(* CODESYS project Лабораторная работа №1.project

Project tree, tasks and I/O mapping:
  Device : CODESYS Control Win V3, 3S - Smart Software Solutions GmbH, order no. 305021, version 3.5.5.50
    application Application
      libraries: Standard, * (System)
      task MainTask (cyclic, interval t#20ms, priority 1) calls PLC_PRG
      task VISU_TASK (cyclic, interval 100 ms, priority 31) calls VisuElems.Visu_Prg
      program PLC_PRG [ST]
      global variables GVL
      visualisation Visualization
  text list GlobalTextList
*)

// Device/Application/GVL
VAR_GLOBAL
	upper_level_sensor: BOOL := FALSE;
	lower_level_sensor: BOOL := FALSE;
	
	pump_relay: BOOL := FALSE;
	yellow_lamp: BOOL := FALSE;
	green_lamp: BOOL := TRUE;
END_VAR

// Device/Application/PLC_PRG
PROGRAM PLC_PRG
VAR
	is_pumping: BOOL := FALSE;
END_VAR

// запускать/останавливать откачку 
// только при срабатывании сенсора
IF upper_level_sensor THEN
	is_pumping := TRUE;
ELSIF lower_level_sensor THEN
	is_pumping := FALSE;
END_IF

// если откачка запущена/остановлена,
// но реле ещё не сработало/отключено,
// то включить/отключить реле и нужную лампочку
IF is_pumping AND NOT pump_relay THEN
	pump_relay := TRUE;
	yellow_lamp := TRUE;
	green_lamp := FALSE;
ELSIF NOT is_pumping AND pump_relay THEN
	pump_relay := FALSE;
	yellow_lamp := FALSE;
	green_lamp := TRUE;
END_IF

END_PROGRAM

// Device/Application/Visualization
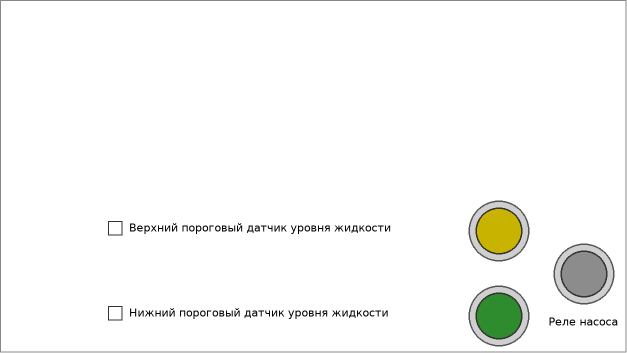
VISUALIZATION Visualization  // 627x353
    Checkbox (106,216 294x24), "Верхний пороговый датчик уровня жидкости", variable: upper_level_sensor
    Checkbox (106,301 294x24), "Нижний пороговый датчик уровня жидкости", variable: lower_level_sensor
    Group (464,196 70x155)
        Lamp1 (0,0 70x70), variable: yellow_lamp, style: Lamp-Lamp1-Yellow
        Lamp1 (0,85 70x70), variable: green_lamp, style: Lamp-Lamp1-Green
    Lamp1 (549,239 70x70), variable: pump_relay, style: Lamp-Lamp1-Gray
    Label (542,307 83x30), "Реле насоса"
END_VISUALIZATION
